// This function has been automatically generated from the project information.
{attribute 'signature_flag' := '1073741824'}
{attribute 'TcGenerated'}
{attribute 'no-analysis'}
FUNCTION F_GetCompany : WSTRING
VAR_INPUT
	
END_VAR

F_GetCompany := "Beckhoff UK";

END_FUNCTION

(* stored: Version 1.1.0.1
   POU F_GetCompany: Id {adf7e1f6-693e-4e58-9bb2-0a8c670647ff}, SpecialFunc None *)
